{attribute 'GeneratedUsingTerminal: EK1122-0000-0018'}
{attribute addProperty BoxType "EK1122-0000-0018"}
{attribute addProperty Id "Beckhoff_EJ3xxxsub_EK1100EK1100_1FC0878B2"}
{attribute addProperty CRC "442345893"}
{attribute addProperty Size "2"}
TYPE Beckhoff_EJ3xxxEK1122_1A5DA9A5 EXTENDS EK1122_1FC0878B :
STRUCT
	{attribute addProperty Name "Beckhoff_EJ3xxxsub_EK1100"}
	{attribute addProperty PreviousPort "Beckhoff EJ3xxxEK1122 : D"}
	Beckhoff_EJ3xxxsub_EK1100 : EK1100_1FC0878B;
END_STRUCT
END_TYPE

(* stored: Version 1.2.0.0, ProductVersion 3.1.4024.9
   DUT Beckhoff_EJ3xxxEK1122_1A5DA9A5: Id {c833bf89-5452-4389-b53c-609ba19178fa} *)
